FUNCTION_BLOCK LC_LT (* Composite Function Block Type *)
  (* Standard: 61499-2 *)
  (* Version 0.0, 2011-08-30, 4DIAC-IDE, 4DIAC-Consortium *)
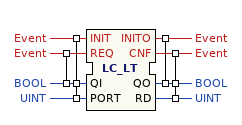
  EVENT_INPUT
    INIT WITH QI, PORT; (* Initialization Request *)
    REQ WITH QI; (* Normal Execution Request *)
  END_EVENT
  EVENT_OUTPUT
    INITO WITH QO; (* Initialization Confirm *)
    CNF WITH QO, RD; (* Execution Confirmation *)
  END_EVENT
  VAR_INPUT
    QI : BOOL; (* Input event qualifier *)
    PORT : UINT; (* Port # *)
  END_VAR
  VAR_OUTPUT
    QO : BOOL; (* Output event qualifier *)
    RD : UINT; (* Read sensor value *)
  END_VAR
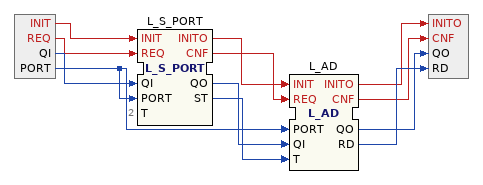
  FBS
    L_S_PORT : L_S_PORT(T := 2);
    L_AD : L_AD;
  END_FBS
  EVENT_CONNECTIONS
    INIT TO L_S_PORT.INIT;
    REQ TO L_S_PORT.REQ;
    L_S_PORT.INITO TO L_AD.INIT;
    L_S_PORT.CNF TO L_AD.REQ;
    L_AD.INITO TO INITO;
    L_AD.CNF TO CNF;
  END_CONNECTIONS
  DATA_CONNECTIONS
    QI TO L_S_PORT.QI;
    PORT TO L_S_PORT.PORT;
    PORT TO L_AD.PORT;
    L_S_PORT.QO TO L_AD.QI;
    L_S_PORT.ST TO L_AD.T;
    L_AD.QO TO QO;
    L_AD.RD TO RD;
  END_CONNECTIONS
END_FUNCTION_BLOCK
